// Creates a Sift Proxy Protocol "ping" Endpoint Message.
FUNCTION _F_CreatePingMessage
VAR_INPUT
	stMsg : REFERENCE TO _ST_SiftMessage;
END_VAR

VAR
	sPingRequest : STRING(255) := '{}';
END_VAR

VAR_OUTPUT
	stErr : ST_SiftError;
END_VAR

stErr := _F_CreateEndpointMessage(sEndpoint := 'ping', 
                                  pData := ADR(sPingRequest), 
                                  nLength := INT_TO_UDINT(LEN(sPingRequest)), 
                                  nBufferLength := 255, 
                                  stMsg := stMsg);

END_FUNCTION

(* stored: Version 1.1.0.1
   POU _F_CreatePingMessage: Id {f66f2735-207d-4dcd-8e50-ed9c5d150534}, SpecialFunc None *)
